KUKA KRL program: ResetaPallet.src, ResetaPallet.dat

--- ResetaPallet.src ---
&ACCESS RVO3
&REL 3
&PARAM EDITMASK = *
DEF ResetaPallet( )
   ;precisa saber qual o pallet ativo
   ;atravez do pallet ativo o programa sabe qual mozaico est� selecionado

   ;FOLD RESETA PALLET
      StrPallet[PalletAtivo].Livre=TRUE
      StrPallet[PalletAtivo].ReceitaAtivo=1
      StrPallet[PalletAtivo].PlaceAtivo=1
      StrPallet[PalletAtivo].CamadaAtiva=1
   ;ENDFOLD

END

--- ResetaPallet.dat ---
DEFDAT  ResetaPallet

ENDDAT
